# EPICS autosave request: 100idPyCRLApp/Db/pyDevCRL_general_settings.req
$(P)$(SYSID):EnergyLocal.VAL
$(P)$(SYSID):EnergySelect.VAL
